FUNCTION_BLOCK OR_88A3DD8EC65DD11C (* Logical OR *)
  (* Standard: 61499-2 *)
  (* Version 1.0, 24.09.2008, marumil, nxtControl GmbH, Initial Version *)
  PACKAGE Main;
  (* Compiler Cpp *)
  {SET_ATTRIBUTE(Runtime.FBType.ImplementingType, Runtime.Standard#DYNGEN_OR)}
  {SET_ATTRIBUTE(Configuration.GenericFBType.InterfaceParams, Runtime.Standard#CNT:=2;OUT:BOOL)}
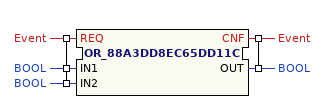
  EVENT_INPUT
    REQ WITH IN1, IN2; (* Normal Execution Request *)
  END_EVENT
  EVENT_OUTPUT
    CNF WITH OUT; (* Execution Confirmation *)
  END_EVENT
  VAR_INPUT
    IN1 : BOOL; (* Argument *)
    IN2 : BOOL; (* Argument *)
  END_VAR
  VAR_OUTPUT
    OUT : BOOL; (* Result: IN1 OR IN2 OR ... *)
  END_VAR
  EC_STATES
    START;
  END_STATES
END_FUNCTION_BLOCK
